(* IEC 61131-3 sources: TSA-FMICS22/ahorn/test/file/se, 27 files *)

(* ---- antivalent_test.st ---- *)
PROGRAM SFAntivalent
 VAR_INPUT
        Activate           : BOOL;
        SChannelNC        : SAFEBOOL;
        SChannelNO        : SAFEBOOL;
        DiscrepancyTime    : TIME;
 END_VAR
 VAR_OUTPUT
        Ready              : BOOL;
        SAntivalentOut    : BOOL;
        Error              : BOOL;
        DiagCode           : WORD;
 END_VAR
 VAR
        Timer1        : TONX;
 END_VAR

IF NOT Activate THEN
    DiagCode := 16#0000;
ELSE

CASE DiagCode OF
16#0000:
    IF Activate THEN
        DiagCode := 16#8001;
    END_IF;
16#8001:
    IF SChannelNC AND SChannelNO THEN
        DiagCode := 16#8004;
        Timer1(IN:=TRUE, PT:=DiscrepancyTime);
    ELSIF NOT SChannelNC AND NOT SChannelNO THEN
        DiagCode := 16#8014;
        Timer1(IN:=TRUE, PT:=DiscrepancyTime);
    ELSIF SChannelNC AND NOT SChannelNO THEN
        DiagCode := 16#8000;
    END_IF;
16#8004:
    IF Timer1.Q THEN
        DiagCode := 16#C001;
    ELSIF NOT SChannelNC THEN
        DiagCode := 16#8001;
    ELSIF NOT SChannelNO THEN
        DiagCode := 16#8000;
    END_IF;
16#C001,
16#C002:
    IF NOT SChannelNC AND SChannelNO THEN
        DiagCode := 16#8001;
    END_IF;
16#8014:
    IF Timer1.Q THEN
        DiagCode := 16#C002;
    ELSIF SChannelNO THEN
        DiagCode := 16#8001;
    ELSIF SChannelNC THEN
        DiagCode := 16#8000;
    END_IF;
16#C003:
    IF NOT SChannelNC AND SChannelNO THEN
        DiagCode := 16#8001;
    END_IF;
16#8005:
    IF Timer1.Q THEN
        DiagCode := 16#C003;
    ELSIF NOT SChannelNC AND SChannelNO THEN
        DiagCode := 16#8001;
    END_IF;
16#8000:
    IF NOT SChannelNC OR SChannelNO THEN
        DiagCode := 16#8005;
        Timer1(IN:=TRUE, PT:=DiscrepancyTime);
    ELSIF NOT SChannelNC AND SChannelNO THEN
        DiagCode := 16#8001;
    END_IF;
END_CASE;
END_IF;

CASE DiagCode OF
16#0000:
    Timer1(IN:=FALSE, PT:=DiscrepancyTime);
    Ready := FALSE;
    Error := FALSE;
    SAntivalentOut:= FALSE;
16#8000:
    Timer1(IN:=FALSE, PT:=DiscrepancyTime);
    Ready := TRUE;
    Error := FALSE;
    SAntivalentOut := TRUE;
16#8001:
    Timer1(IN:=FALSE, PT:=DiscrepancyTime);
    Ready := TRUE;
    Error := FALSE;
    SAntivalentOut:= FALSE;
16#8004,
16#8014,
16#8005:
	Timer1(IN:=TRUE, PT:=DiscrepancyTime);
    Ready := TRUE;
    Error := FALSE;
    SAntivalentOut:= FALSE;
16#C001,
16#C002,
16#C003:
    Timer1(IN:=FALSE, PT:=DiscrepancyTime);
    Ready := TRUE;
    Error := TRUE;
    SAntivalentOut:= FALSE;
END_CASE;

END_PROGRAM

FUNCTION_BLOCK TONX
VAR_INPUT
  IN : BOOL;
  PT : TIME;
END_VAR
VAR
  running : BOOL;
END_VAR
VAR_TEMP
    timeout : BOOL;
END_VAR
VAR_OUTPUT
  Q : BOOL;
  ET : TIME;
END_VAR

  timeout := NONDETERMINISTIC_BOOL();

  IF NOT IN THEN
    Q := FALSE;
    running := FALSE;
  ELSIF NOT running AND NOT Q THEN
    running := TRUE;
  ELSIF running AND NOT Q THEN
    Q := timeout;
    running := NOT Q;
  END_IF;

  ET := NONDETERMINISTIC_TIME();
END_FUNCTION_BLOCK

(* ---- call.st ---- *)
PROGRAM P
VAR_INPUT
    x : INT;
END_VAR
VAR
    f : Fb;
END_VAR
VAR_OUTPUT
    y : INT;
END_VAR
    f(a:=x,b=>y);
END_PROGRAM

FUNCTION_BLOCK Fb
VAR_INPUT
    a : INT;
END_VAR
VAR_OUTPUT
    b : INT;
END_VAR;
    IF a >= 32 THEN
        b := 64;
    ELSE
        b := 16;
    END_IF;
END_FUNCTION_BLOCK

(* ---- call_coverage_in_1_cycle_with_change_shadow.st ---- *)
PROGRAM P
VAR_INPUT
    a : INT;
END_VAR
VAR
    f : Fb;
END_VAR
VAR_OUTPUT
    b : BOOL;
END_VAR
    f(x:=a,z=>b);
END_PROGRAM

FUNCTION_BLOCK Fb
VAR_INPUT
    x : INT;
END_VAR
VAR
    y : INT;
END_VAR
VAR_OUTPUT
    z : BOOL;
END_VAR;
    IF x >= 32 THEN
        y := y + change(1, 3);
    ELSE
        y := y;
    END_IF;
    IF y >= 3 THEN
        z := TRUE;
        y := 0;
    ELSE
        z := FALSE;
    END_IF;
END_FUNCTION_BLOCK

(* ---- call_coverage_in_3_cycles.st ---- *)
PROGRAM P
VAR_INPUT
    a : INT;
END_VAR
VAR
    f : Fb;
END_VAR
VAR_OUTPUT
    b : BOOL;
END_VAR
    f(x:=a,z=>b);
END_PROGRAM

FUNCTION_BLOCK Fb
VAR_INPUT
    x : INT;
END_VAR
VAR
    y : INT;
END_VAR
VAR_OUTPUT
    z : BOOL;
END_VAR;
    IF x >= 32 THEN
        y := y + 1;
    ELSE
        y := y;
    END_IF;
    IF y >= 3 THEN
        z := TRUE;
        y := 0;
    ELSE
        z := FALSE;
    END_IF;
END_FUNCTION_BLOCK

(* ---- call_two_times.st ---- *)
PROGRAM P
VAR_INPUT
    x : INT;
END_VAR
VAR
    f : Fb;
END_VAR
VAR_OUTPUT
    y : INT;
END_VAR
    f(a:=x,b=>y);
    f(a:=x,b=>y);
END_PROGRAM

FUNCTION_BLOCK Fb
VAR_INPUT
    a : INT;
END_VAR
VAR_OUTPUT
    b : INT;
END_VAR;
    IF a >= 32 THEN
        b := 64;
    ELSE
        b := 16;
    END_IF;
END_FUNCTION_BLOCK

(* ---- call_with_state.st ---- *)
PROGRAM P
VAR_INPUT
    x : INT;
END_VAR
VAR
    f : Fb;
END_VAR
VAR_OUTPUT
    y : INT;
END_VAR
    f(a:=x,c=>y);
END_PROGRAM

FUNCTION_BLOCK Fb
VAR_INPUT
    a : INT;
END_VAR
VAR
    b : INT;
END_VAR
VAR_OUTPUT
    c : INT;
END_VAR;
    IF a >= 32 THEN
        b := b + 1;
    ELSE
        b := b;
    END_IF;
    c := b;
END_FUNCTION_BLOCK

(* ---- call_with_stateful_if.st ---- *)
PROGRAM P
VAR_INPUT
    x : BOOL;
END_VAR
VAR
    f : Fb;
END_VAR
VAR_OUTPUT
    y : BOOL;
END_VAR
    f(a:=x,c=>y);
END_PROGRAM

FUNCTION_BLOCK Fb
VAR_INPUT
    a : BOOL;
END_VAR
VAR
    b : INT;
END_VAR
VAR_OUTPUT
    c : BOOL;
END_VAR;
    IF a THEN
        b := b + 1;
    ELSE
        b := b;
    END_IF;
    IF b > 3 THEN
        c := TRUE;
        b := 0;
    ELSE
        c := FALSE;
    END_IF;
END_FUNCTION_BLOCK

(* ---- call_with_tripple_diamond.st ---- *)
PROGRAM P
VAR_INPUT
    x : INT;
END_VAR
VAR
    f : Fb;
END_VAR
VAR_OUTPUT
    y : INT;
END_VAR
    f(a:=x,b=>y);
END_PROGRAM

FUNCTION_BLOCK Fb
VAR_INPUT
    a : INT;
END_VAR
VAR_OUTPUT
    b : INT;
END_VAR;
    IF a >= 32 THEN
        b := 64;
    ELSE
        b := 16;
    END_IF;
    IF a >= 32 THEN
        b := 64;
    ELSE
        b := 16;
    END_IF;
    IF a >= 32 THEN
        b := 64;
    ELSE
        b := 16;
    END_IF;
END_FUNCTION_BLOCK

(* ---- dependant_on_call.st ---- *)
PROGRAM P
VAR_INPUT
    x : INT;
END_VAR
VAR
    f : Fb;
END_VAR
VAR
    y : INT;
END_VAR
VAR_OUTPUT
    z : BOOL;
END_VAR
    f(a:=x,b=>y);
    IF y == 64 THEN
        z := TRUE;
    ELSE
        z := FALSE;
    END_IF;
END_PROGRAM

FUNCTION_BLOCK Fb
VAR_INPUT
    a : INT;
END_VAR
VAR_OUTPUT
    b : INT;
END_VAR;
    IF a >= 32 THEN
        b := 64;
    ELSE
        b := 16;
    END_IF;
END_FUNCTION_BLOCK

(* ---- different_frame_stacks.st ---- *)
PROGRAM P
VAR_INPUT
    x : INT;
END_VAR
VAR
    f : Fb1;
    g : Fb2;
    y : BOOL;
END_VAR
VAR_OUTPUT
    z : BOOL;
END_VAR
    IF x >= 32 THEN
        f(a:=16,b=>y);
    ELSE
        g(a:=0,b=>y);
    END_IF;
    IF y THEN
        z := TRUE;
    ELSE
        z := FALSE;
    END_IF;
END_PROGRAM

FUNCTION_BLOCK Fb1
VAR_INPUT
    a : INT;
END_VAR
VAR
    h : Fb3;
END_VAR
VAR_OUTPUT
    b : BOOL;
END_VAR;
    h(a:=a,b=>b);
    IF a >= 16 THEN
        b := TRUE;
    ELSE
        b := FALSE;
    END_IF;
END_FUNCTION_BLOCK

FUNCTION_BLOCK Fb2
VAR_INPUT
    a : INT;
END_VAR
VAR
    h : Fb3;
END_VAR
VAR_OUTPUT
    b : BOOL;
END_VAR;
    h(a:=a,b=>b);
    IF a >= 16 THEN
        b := TRUE;
    ELSE
        b := FALSE;
    END_IF;
END_FUNCTION_BLOCK

FUNCTION_BLOCK Fb3
VAR_INPUT
    a : INT;
END_VAR
VAR_OUTPUT
    b : BOOL;
END_VAR;
    IF a >= 16 THEN
        b := TRUE;
    ELSE
        b := FALSE;
    END_IF;
    b := FALSE;
END_FUNCTION_BLOCK

(* ---- emergency_stop_test.st ---- *)
PROGRAM SFEmergencyStop2
VAR_INPUT
        Activate      : BOOL;
        SEStopIn     : BOOL;
        SStartReset  : BOOL;
        SAutoReset   : BOOL;
        Reset         : BOOL;
 END_VAR

 VAR_OUTPUT
        Ready         : BOOL;
        SEStopOut    : BOOL;
        Error         : BOOL;
        DiagCode      : WORD;
 END_VAR

 VAR
        RTRIGatReset: R_TRIG;
 END_VAR

RTRIGatReset(CLK:=Reset);

IF NOT Activate THEN
    DiagCode := 16#0000;
ELSE

CASE DiagCode OF
16#0000:
    IF Activate THEN
        DiagCode := 16#8001;
    END_IF;
16#8001:
    IF NOT SStartReset THEN
        DiagCode := 16#8002;
    ELSIF SStartReset AND NOT SEStopIn THEN
        DiagCode := 16#8004;
    ELSIF SEStopIn AND SStartReset THEN
        DiagCode := 16#8000;
    END_IF;
16#8002:
    IF SEStopIn THEN
        DiagCode := 16#8003;
    END_IF;
16#8003:
    IF Reset AND NOT RTRIGatReset.Q THEN
        DiagCode := 16#C001;
    ELSIF NOT SEStopIn THEN
        DiagCode := 16#8002;
    ELSIF RTRIGatReset.Q THEN
        DiagCode := 16#8000;
    END_IF;
16#C001:
    IF NOT Reset THEN
        DiagCode := 16#8003;
    END_IF;
16#8004:
    IF SEStopIn AND NOT SAutoReset THEN
        DiagCode := 16#8005;
    ELSIF SEStopIn AND SAutoReset THEN
        DiagCode := 16#8000;
    END_IF;
16#8005:
    IF Reset AND NOT RTRIGatReset.Q THEN
        DiagCode := 16#C002;
    ELSIF NOT SEStopIn THEN
        DiagCode := 16#8004;
    ELSIF RTRIGatReset.Q OR SAutoReset THEN
        DiagCode := 16#8000;
    END_IF;
16#C002:
    IF NOT Reset THEN
        DiagCode := 16#8005;
    END_IF;
16#8000:
    IF NOT SEStopIn THEN
        DiagCode := 16#8004;
    END_IF;
END_CASE;
END_IF;

CASE DiagCode OF
16#0000:
    Ready := FALSE;
    Error := FALSE;
    SEStopOut := FALSE;
16#8001:
    Ready := TRUE;
    Error := FALSE;
    SEStopOut := FALSE;
16#8002:
    Ready := TRUE;
    Error := FALSE;
    SEStopOut := FALSE;
16#8003:
    Ready := TRUE;
    Error := FALSE;
    SEStopOut := FALSE;
16#C001:
    Ready := TRUE;
    Error := TRUE;
    SEStopOut := FALSE;
16#8004:
    Ready := TRUE;
    Error := FALSE;
    SEStopOut := FALSE;
16#8005:
    Ready := TRUE;
    Error := FALSE;
    SEStopOut := FALSE;
16#C002:
    Ready := TRUE;
    Error := TRUE;
    SEStopOut := FALSE;
16#8000:
    Ready := TRUE;
    Error := FALSE;
    SEStopOut := TRUE;
END_CASE;

END_PROGRAM

FUNCTION_BLOCK R_TRIG
VAR_INPUT
   CLK: BOOL;
END_VAR
VAR_OUTPUT
   Q: BOOL;
END_VAR
VAR
   M: BOOL;
END_VAR
Q := CLK AND NOT M;
M := CLK;
END_FUNCTION_BLOCK

(* ---- merge_if_call.st ---- *)
PROGRAM P
VAR_INPUT
    x : INT;
END_VAR
VAR
    f : Fb;
    y : BOOL;
END_VAR
VAR_OUTPUT
    z : BOOL;
END_VAR
    IF x >= 32 THEN
        f(a:=16,b=>y);
    ELSE
        f(a:=0,b=>y);
    END_IF;
    IF y THEN
        z := TRUE;
    ELSE
        z := FALSE;
    END_IF;
END_PROGRAM

FUNCTION_BLOCK Fb
VAR_INPUT
    a : INT;
END_VAR
VAR_OUTPUT
    b : BOOL;
END_VAR;
    IF a >= 16 THEN
        b := TRUE;
    ELSE
        b := FALSE;
    END_IF;
END_FUNCTION_BLOCK

(* ---- assignment.st ---- *)
PROGRAM P
VAR
    x : INT;
END_VAR
    x := x + 1;
END_PROGRAM

(* ---- branch_coverage_in_3_cycles.st ---- *)
PROGRAM P
VAR_INPUT
    x : INT;
END_VAR
VAR
    y : INT;
    z : BOOL;
END_VAR
    IF x >= 32 THEN
        y := y + 1;
    ELSE
        y := y;
    END_IF;
    IF y >= 3 THEN
        z := TRUE;
        y := 0;
    ELSE
        z := FALSE;
    END_IF;
END_PROGRAM

(* ---- breadth-first_and_merging.st ---- *)
PROGRAM P
VAR_INPUT
    x : INT;
    y : INT;
END_VAR
VAR
    a : INT;
    b : BOOL;
END_VAR
    IF x <= 128 THEN
        a := a + 1;
        IF y <= 128 THEN
            IF x <= 64 THEN
                IF x <= 32 THEN
                    a := 1;
                ELSE
                    a := 2;
                END_IF;
            ELSE
                IF x <= 96 THEN
                    a := 3;
                ELSE
                    a := 4;
                END_IF;
                a := a + a;
            END_IF;
        ELSE
            a := 0;
        END_IF;
        a := a + 1;
    ELSE
        a := a;
    END_IF;
    IF a >= 3 THEN
        b := TRUE;
        a := 0;
    ELSE
        b := FALSE;
    END_IF;
END_PROGRAM

(* ---- constant_propagation.st ---- *)
PROGRAM P
VAR
    x : INT;
    y : INT;
    z : INT;
END_VAR
    x := x + 1;
    y := 2;
    z := x + y;
END_PROGRAM

(* ---- constant_propagation_with_input.st ---- *)
PROGRAM P
VAR_INPUT
    a : INT;
END_VAR
VAR
    x : INT;
    y : INT;
    z : INT;
END_VAR
    x := x + 1 - a;
    y := 2;
    z := x + y;
END_PROGRAM

(* ---- constant_propagation_with_shadows.st ---- *)
PROGRAM P
VAR
    x : INT;
    y : INT;
    z : INT;
END_VAR
    x := x + change(0, 1);
    y := change(y, 2);
    z := x + y;
END_PROGRAM

(* ---- if.st ---- *)
PROGRAM P
VAR_INPUT
    x : INT;
END_VAR
VAR
    y : BOOL;
END_VAR
    IF x >= 32 THEN
        y := TRUE;
    ELSE
        y := FALSE;
    END_IF;
END_PROGRAM

(* ---- if_change.st ---- *)
PROGRAM P
VAR
    x : BOOL;
END_VAR
    IF change(TRUE, FALSE) THEN
        x := TRUE;
    ELSE
        x := FALSE;
    END_IF;
END_PROGRAM

(* ---- if_reaching_change.st ---- *)
PROGRAM P
VAR
    x : INT;
    y : INT;
    z : BOOL;
END_VAR
    x := 1 + change(y, y + 1);
    IF (y + 1) = x THEN
        z := TRUE;
    ELSE
        z := FALSE;
    END_IF;
END_PROGRAM

(* ---- if_with_state.st ---- *)
PROGRAM P
VAR_INPUT
    x : INT;
END_VAR
VAR
    y : INT;
END_VAR
    IF x >= 32 THEN
        y := y + 1;
    ELSE
        y := y;
    END_IF;
END_PROGRAM

(* ---- mode_selector_test.st ---- *)
PROGRAM ModeSelectorX
VAR_INPUT
        Activate        : BOOL;
        SMode0         : BOOL;
        SMode1         : BOOL;
        SMode2         : BOOL;
        SMode3         : BOOL;
        SMode4         : BOOL;
        SMode5         : BOOL;
        SMode6         : BOOL;
        SMode7         : BOOL;
        SUnlock        : BOOL;
        SSetMode       : BOOL;
        AutoSetMode     : BOOL;
        ModeMonitorTime : TIME;
        Reset           : BOOL;
 END_VAR
 VAR_OUTPUT
        Ready           : BOOL;
        SMode0Sel      : BOOL;
        SMode1Sel      : BOOL;
        SMode2Sel      : BOOL;
        SMode3Sel      : BOOL;
        SMode4Sel      : BOOL;
        SMode5Sel      : BOOL;
        SMode6Sel      : BOOL;
        SMode7Sel      : BOOL;
        SAnyModeSel    : BOOL;
        Error           : BOOL;
        DiagCode        : WORD;
 END_VAR
 VAR
        Timer1        : TONX;                 (* Timer for S2, transition T27 *)
 END_VAR

 VAR
        RTRIGatReset: RTRIG;
        RTRIGatSetMode: RTRIG;
        FTRIGatModeSel0: FTRIG;
        RTRIGatModeSel0: RTRIG;
        fallingEdgeDetected : BOOL;
 END_VAR

 VAR_TEMP
    Error1 : BOOL;
    Error2 : BOOL;
 END_VAR

RTRIGatReset(CLK:=Reset);
RTRIGatSetMode(CLK:=SSetMode);

IF NOT Activate THEN
    DiagCode := 16#0000;
ELSE

IF (SMode0 OR SMode1 OR SMode2 OR SMode3 OR SMode4 OR SMode5 OR SMode6 OR SMode7) AND NOT ((
                                                                                                  (NOT SMode0 AND NOT SMode1 AND NOT SMode2 AND NOT SMode3 AND NOT SMode4 AND NOT SMode5 AND NOT SMode6 AND SMode7) OR
                                                                                                  (NOT SMode0 AND NOT SMode1 AND NOT SMode2 AND NOT SMode3 AND NOT SMode4 AND NOT SMode5 AND SMode6 AND NOT SMode7) OR
                                                                                                  (NOT SMode0 AND NOT SMode1 AND NOT SMode2 AND NOT SMode3 AND NOT SMode4 AND SMode5 AND NOT SMode6 AND NOT SMode7) OR
                                                                                                  (NOT SMode0 AND NOT SMode1 AND NOT SMode2 AND NOT SMode3 AND SMode4 AND NOT SMode5 AND NOT SMode6 AND NOT SMode7) OR
                                                                                                  (NOT SMode0 AND NOT SMode1 AND NOT SMode2 AND SMode3 AND NOT SMode4 AND NOT SMode5 AND NOT SMode6 AND NOT SMode7) OR
                                                                                                  (NOT SMode0 AND NOT SMode1 AND SMode2 AND NOT SMode3 AND NOT SMode4 AND NOT SMode5 AND NOT SMode6 AND NOT SMode7) OR
                                                                                                  (NOT SMode0 AND SMode1 AND NOT SMode2 AND NOT SMode3 AND NOT SMode4 AND NOT SMode5 AND NOT SMode6 AND NOT SMode7) OR
                                                                                                  (SMode0 AND NOT SMode1 AND NOT SMode2 AND NOT SMode3 AND NOT SMode4 AND NOT SMode5 AND NOT SMode6 AND NOT SMode7))) THEN
    Error1 := true;
ELSE
    Error1 := false;
END_IF;

CASE DiagCode OF
16#0000:
    IF Activate THEN
        DiagCode := 16#8005;
    END_IF;
16#8005:
    IF (NOT SMode0 AND NOT SMode1 AND NOT SMode2 AND NOT SMode3 AND NOT SMode4 AND NOT SMode5 AND NOT SMode6 AND NOT SMode7) THEN
        FTRIGatModeSel0(CLK:=false);
        RTRIGatModeSel0(CLK:=false);
    ELSE
        FTRIGatModeSel0(CLK:=true);
        RTRIGatModeSel0(CLK:=true);
    END_IF;

    IF FTRIGatModeSel0.Q THEN
        fallingEdgeDetected := TRUE;
    END_IF;

    IF fallingEdgeDetected THEN
        Timer1(IN:=true, PT:=ModeMonitorTime);
    ELSIF RTRIGatModeSel0.Q THEN
        Timer1(IN:=false, PT:=ModeMonitorTime);
        fallingEdgeDetected := FALSE;
    END_IF;

    Error2 := Timer1.Q;

    IF Error1 THEN
        DiagCode := 16#C001;
    ELSIF Error2 THEN
        DiagCode := 16#C002;
    ELSIF ((AutoSetMode OR RTRIGatSetMode.Q) AND SUnlock AND ((NOT SMode0 AND NOT SMode1 AND NOT SMode2 AND NOT SMode3 AND NOT SMode4 AND NOT SMode5 AND NOT SMode6 AND SMode7) OR
                                                               (NOT SMode0 AND NOT SMode1 AND NOT SMode2 AND NOT SMode3 AND NOT SMode4 AND NOT SMode5 AND SMode6 AND NOT SMode7) OR
                                                               (NOT SMode0 AND NOT SMode1 AND NOT SMode2 AND NOT SMode3 AND NOT SMode4 AND SMode5 AND NOT SMode6 AND NOT SMode7) OR
                                                               (NOT SMode0 AND NOT SMode1 AND NOT SMode2 AND NOT SMode3 AND SMode4 AND NOT SMode5 AND NOT SMode6 AND NOT SMode7) OR
                                                               (NOT SMode0 AND NOT SMode1 AND NOT SMode2 AND SMode3 AND NOT SMode4 AND NOT SMode5 AND NOT SMode6 AND NOT SMode7) OR
                                                               (NOT SMode0 AND NOT SMode1 AND SMode2 AND NOT SMode3 AND NOT SMode4 AND NOT SMode5 AND NOT SMode6 AND NOT SMode7) OR
                                                               (NOT SMode0 AND SMode1 AND NOT SMode2 AND NOT SMode3 AND NOT SMode4 AND NOT SMode5 AND NOT SMode6 AND NOT SMode7) OR
                                                               (SMode0 AND NOT SMode1 AND NOT SMode2 AND NOT SMode3 AND NOT SMode4 AND NOT SMode5 AND NOT SMode6 AND NOT SMode7))) THEN
        DiagCode := 16#8000;
    END_IF;
16#8000:
    IF Error1 THEN
        DiagCode := 16#C001;
    ELSIF (SMode0 <> SMode0Sel OR SMode1 <> SMode1Sel OR SMode2 <> SMode2Sel OR SMode3 <> SMode3Sel
          OR SMode4 <> SMode4Sel OR SMode5 <> SMode5Sel OR SMode6 <> SMode6Sel OR SMode7 <> SMode7Sel) THEN
        DiagCode := 16#8005;
        fallingEdgeDetected := FALSE;
    ELSIF (NOT SUnlock) THEN
        DiagCode := 16#8004;
    END_IF;
16#8004:
    IF SUnlock THEN
        DiagCode := 16#8000;
    END_IF;
16#C001:
    IF Reset AND NOT RTRIGatReset.Q THEN
        DiagCode := 16#C003;
    ELSIF RTRIGatReset.Q THEN
        DiagCode := 16#8005;
        fallingEdgeDetected := FALSE;
    END_IF;
16#C002:
    IF Reset AND NOT RTRIGatReset.Q THEN
        DiagCode := 16#C004;
    ELSIF RTRIGatReset.Q THEN
        DiagCode := 16#8005;
        fallingEdgeDetected := FALSE;
    END_IF;
16#C003:
    IF (NOT Reset) THEN
                DiagCode := 16#C001;
    END_IF;
16#C004:
    IF (NOT Reset) THEN
                DiagCode := 16#C002;
    END_IF;
END_CASE;
END_IF;

CASE DiagCode OF
16#0000:
    Ready := false;
    SMode0Sel := false;
    SMode1Sel := false;
    SMode2Sel := false;
    SMode3Sel := false;
    SMode4Sel := false;
    SMode5Sel := false;
    SMode6Sel := false;
    SMode7Sel := false;
    SAnyModeSel := false;
    Error := false;
16#8005:
    Ready := true;
    SMode0Sel := false;
    SMode1Sel := false;
    SMode2Sel := false;
    SMode3Sel := false;
    SMode4Sel := false;
    SMode5Sel := false;
    SMode6Sel := false;
    SMode7Sel := false;
    SAnyModeSel := false;
    Error := false;
16#8000:
    Ready := true;
    SMode0Sel := SMode0;
    SMode1Sel := SMode1;
    SMode2Sel := SMode2;
    SMode3Sel := SMode3;
    SMode4Sel := SMode4;
    SMode5Sel := SMode5;
    SMode6Sel := SMode6;
    SMode7Sel := SMode7;
    SAnyModeSel := true;
    Error := false;
16#8004:
    Ready := true;
    SAnyModeSel := true;
    Error := false;
16#C001,
16#C002,
16#C003,
16#C004:
    Ready := true;
    SMode0Sel := false;
    SMode1Sel := false;
    SMode2Sel := false;
    SMode3Sel := false;
    SMode4Sel := false;
    SMode5Sel := false;
    SMode6Sel := false;
    SMode7Sel := false;
    SAnyModeSel := false;
    Error := true;
END_CASE;

IF (DiagCode <> 16#8005) THEN
    Timer1(IN:=false, PT:=ModeMonitorTime);
END_IF;
END_PROGRAM

FUNCTION_BLOCK TONX
VAR_INPUT
  IN : BOOL;
  PT : TIME;
END_VAR
VAR
  running : BOOL;
END_VAR
VAR_TEMP
    timeout : BOOL;
END_VAR
VAR_OUTPUT
  Q : BOOL;
  ET : TIME;
END_VAR

  timeout := NONDETERMINISTIC_BOOL();

  IF NOT IN THEN
    Q := FALSE;
    running := FALSE;
  ELSIF NOT running AND NOT Q THEN
    running := TRUE;
  ELSIF running AND NOT Q THEN
    Q := timeout;
    running := NOT Q;
  END_IF;

  ET := NONDETERMINISTIC_TIME();
END_FUNCTION_BLOCK

FUNCTION_BLOCK RTRIG
VAR_INPUT
   CLK: BOOL;
END_VAR
VAR_OUTPUT
   Q: BOOL;
END_VAR
VAR
   M: BOOL;
END_VAR
Q := CLK AND NOT M;
M := CLK;
END_FUNCTION_BLOCK

FUNCTION_BLOCK FTRIG
VAR_INPUT
   CLK: BOOL;
END_VAR
VAR_OUTPUT
   Q: BOOL;
END_VAR
VAR
   M: BOOL;
END_VAR
Q := NOT CLK AND M;
M := CLK;
END_FUNCTION_BLOCK

(* ---- non_deterministic_if.st ---- *)
PROGRAM P
VAR
    x : BOOL;
    y : BOOL;
END_VAR
    x := NONDETERMINISTIC_BOOL();
    IF x THEN
        y := TRUE;
    ELSE
        y := FALSE;
    END_IF;
END_PROGRAM

(* ---- unreachable_if.st ---- *)
PROGRAM P
VAR
    y : BOOL;
END_VAR
    IF FALSE THEN
        y := TRUE;
    ELSE
        y := FALSE;
    END_IF;
END_PROGRAM

(* ---- while.st ---- *)
PROGRAM P
VAR
    x : INT;
    y : INT;
END_VAR
    x := 1;
    y := 0;
    WHILE y > 0 DO
        x := x + y;
        y := y + 1;
    END_WHILE;
END_PROGRAM

(* ---- while_with_if.st ---- *)
PROGRAM P
VAR_INPUT
    y : INT;
    n : INT;
END_VAR
VAR
    x : INT;
END_VAR
    x := 0;
    WHILE x < n DO
        IF y > 0 THEN
            x := x + y;
        ELSE
            x := x - y;
        END_IF;
        y := -1 * y;
    END_WHILE;
END_PROGRAM
